FUNCTION_BLOCK IntegerSchreiben
VAR_INPUT
	Value: INT;
END_VAR
VAR_OUTPUT
	LowByte: BYTE;
	HighByte: BYTE;
END_VAR
VAR	
END_VAR

LowByte := INT_TO_BYTE(Value);
HighByte := INT_TO_BYTE(Value / 256);

END_FUNCTION_BLOCK

(* stored: Version 1.1.0.1, ProductVersion 3.1.4024.5
   POU IntegerSchreiben: Id {e01eaed2-b029-4252-a378-1f0bb01560d3}, SpecialFunc None *)
